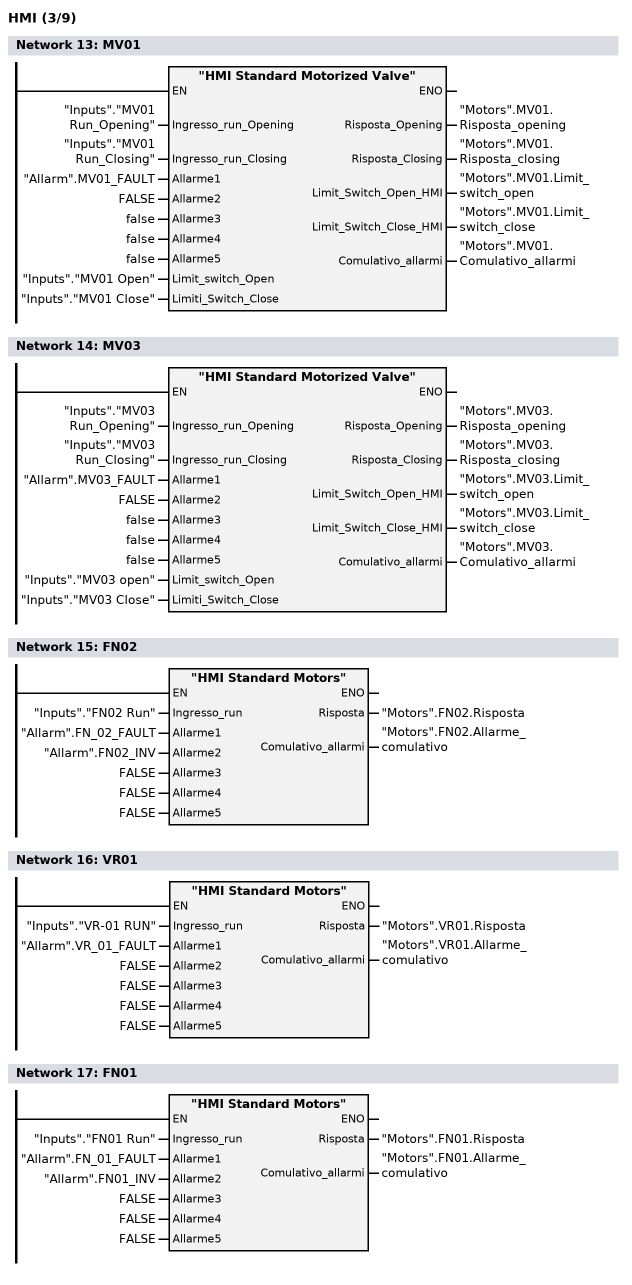
   RUNG wire#powerrail
      "HMI Standard Motorized Valve"(Ingresso_run_Opening := "Inputs"."MV01 Run_Opening", Ingresso_run_Closing := "Inputs"."MV01 Run_Closing", Allarme1 := "Allarm".MV01_FAULT, Allarme2 := FALSE, Allarme3 := false, Allarme4 := false, Allarme5 := false, Limit_switch_Open := "Inputs"."MV01 Open", Limiti_Switch_Close := "Inputs"."MV01 Close", Risposta_Opening => "Motors".MV01.Risposta_opening, Risposta_Closing => "Motors".MV01.Risposta_closing, Limit_Switch_Open_HMI => "Motors".MV01.Limit_switch_open, Limit_Switch_Close_HMI => "Motors".MV01.Limit_switch_close, Comulativo_allarmi => "Motors".MV01.Comulativo_allarmi)
   END_RUNG
   // the same network as SCL:
   "HMI Standard Motorized Valve"(Ingresso_run_Opening := "Inputs"."MV01 Run_Opening",
                           Ingresso_run_Closing := "Inputs"."MV01 Run_Closing",
                           Allarme1 := "Allarm".MV01_FAULT,
                           Allarme2 := FALSE,
                           Allarme3 := false,
                           Allarme4 := false,
                           Allarme5 := false,
                           Limit_switch_Open := "Inputs"."MV01 Open",
                           Limiti_Switch_Close := "Inputs"."MV01 Close",
                           Risposta_Opening => "Motors".MV01.Risposta_opening,
                           Risposta_Closing => "Motors".MV01.Risposta_closing,
                           Limit_Switch_Open_HMI => "Motors".MV01.Limit_switch_open,
                           Limit_Switch_Close_HMI => "Motors".MV01.Limit_switch_close,
                           Comulativo_allarmi => "Motors".MV01.Comulativo_allarmi);
END_REGION

REGION Network 14: MV03
   RUNG wire#powerrail
      "HMI Standard Motorized Valve"(Ingresso_run_Opening := "Inputs"."MV03 Run_Opening", Ingresso_run_Closing := "Inputs"."MV03 Run_Closing", Allarme1 := "Allarm".MV03_FAULT, Allarme2 := FALSE, Allarme3 := false, Allarme4 := false, Allarme5 := false, Limit_switch_Open := "Inputs"."MV03 open", Limiti_Switch_Close := "Inputs"."MV03 Close", Risposta_Opening => "Motors".MV03.Risposta_opening, Risposta_Closing => "Motors".MV03.Risposta_closing, Limit_Switch_Open_HMI => "Motors".MV03.Limit_switch_open, Limit_Switch_Close_HMI => "Motors".MV03.Limit_switch_close, Comulativo_allarmi => "Motors".MV03.Comulativo_allarmi)
   END_RUNG
   // the same network as SCL:
   "HMI Standard Motorized Valve"(Ingresso_run_Opening := "Inputs"."MV03 Run_Opening",
                           Ingresso_run_Closing := "Inputs"."MV03 Run_Closing",
                           Allarme1 := "Allarm".MV03_FAULT,
                           Allarme2 := FALSE,
                           Allarme3 := false,
                           Allarme4 := false,
                           Allarme5 := false,
                           Limit_switch_Open := "Inputs"."MV03 open",
                           Limiti_Switch_Close := "Inputs"."MV03 Close",
                           Risposta_Opening => "Motors".MV03.Risposta_opening,
                           Risposta_Closing => "Motors".MV03.Risposta_closing,
                           Limit_Switch_Open_HMI => "Motors".MV03.Limit_switch_open,
                           Limit_Switch_Close_HMI => "Motors".MV03.Limit_switch_close,
                           Comulativo_allarmi => "Motors".MV03.Comulativo_allarmi);
END_REGION

REGION Network 15: FN02
   RUNG wire#powerrail
      "HMI Standard Motors"(Ingresso_run := "Inputs"."FN02 Run", Allarme1 := "Allarm".FN_02_FAULT, Allarme2 := "Allarm".FN02_INV, Allarme3 := FALSE, Allarme4 := FALSE, Allarme5 := FALSE, Risposta => "Motors".FN02.Risposta, Comulativo_allarmi => "Motors".FN02.Allarme_comulativo)
   END_RUNG
   // the same network as SCL:
   "HMI Standard Motors"(Ingresso_run := "Inputs"."FN02 Run",
                         Allarme1 := "Allarm".FN_02_FAULT,
                         Allarme2 := "Allarm".FN02_INV,
                         Allarme3 := FALSE,
                         Allarme4 := FALSE,
                         Allarme5 := FALSE,
                         Risposta => "Motors".FN02.Risposta,
                         Comulativo_allarmi => "Motors".FN02.Allarme_comulativo);
END_REGION

REGION Network 16: VR01
   RUNG wire#powerrail
      "HMI Standard Motors"(Ingresso_run := "Inputs"."VR-01 RUN", Allarme1 := "Allarm".VR_01_FAULT, Allarme2 := FALSE, Allarme3 := FALSE, Allarme4 := FALSE, Allarme5 := FALSE, Risposta => "Motors".VR01.Risposta, Comulativo_allarmi => "Motors".VR01.Allarme_comulativo)
   END_RUNG
   // the same network as SCL:
   "HMI Standard Motors"(Ingresso_run := "Inputs"."VR-01 RUN",
                         Allarme1 := "Allarm".VR_01_FAULT,
                         Allarme2 := FALSE,
                         Allarme3 := FALSE,
                         Allarme4 := FALSE,
                         Allarme5 := FALSE,
                         Risposta => "Motors".VR01.Risposta,
                         Comulativo_allarmi => "Motors".VR01.Allarme_comulativo);
END_REGION

REGION Network 17: FN01
   RUNG wire#powerrail
      "HMI Standard Motors"(Ingresso_run := "Inputs"."FN01 Run", Allarme1 := "Allarm".FN_01_FAULT, Allarme2 := "Allarm".FN01_INV, Allarme3 := FALSE, Allarme4 := FALSE, Allarme5 := FALSE, Risposta => "Motors".FN01.Risposta, Comulativo_allarmi => "Motors".FN01.Allarme_comulativo)
   END_RUNG
   // the same network as SCL:
   "HMI Standard Motors"(Ingresso_run := "Inputs"."FN01 Run",
                         Allarme1 := "Allarm".FN_01_FAULT,
                         Allarme2 := "Allarm".FN01_INV,
                         Allarme3 := FALSE,
                         Allarme4 := FALSE,
                         Allarme5 := FALSE,
                         Risposta => "Motors".FN01.Risposta,
                         Comulativo_allarmi => "Motors".FN01.Allarme_comulativo);
END_REGION

REGION Network 18: VR02
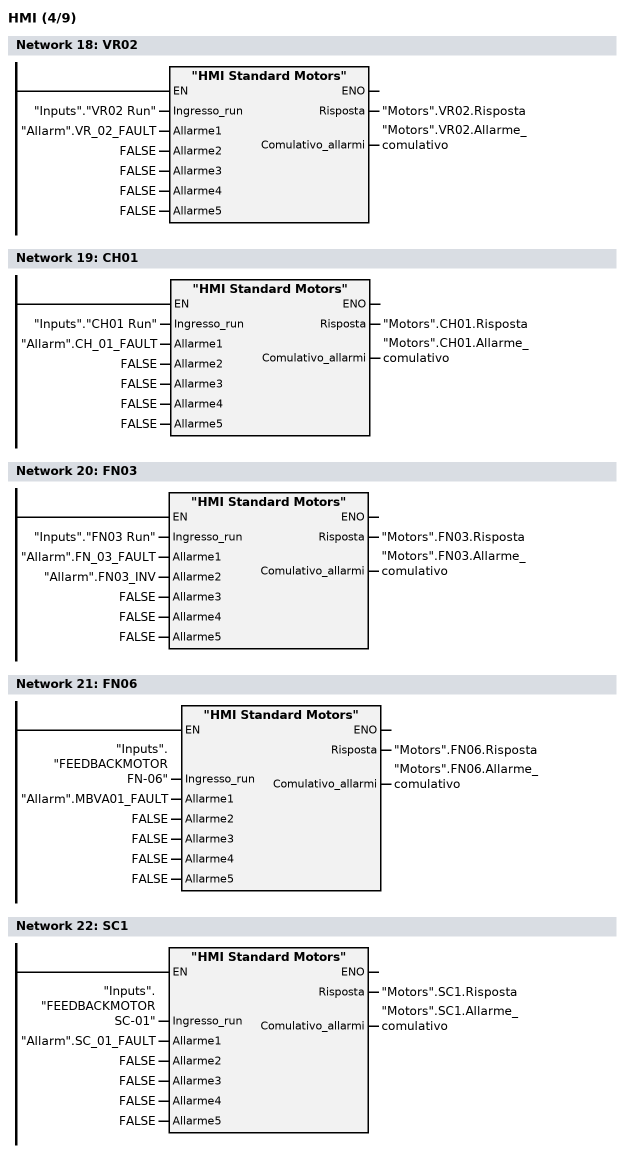
   RUNG wire#powerrail
      "HMI Standard Motors"(Ingresso_run := "Inputs"."VR02 Run", Allarme1 := "Allarm".VR_02_FAULT, Allarme2 := FALSE, Allarme3 := FALSE, Allarme4 := FALSE, Allarme5 := FALSE, Risposta => "Motors".VR02.Risposta, Comulativo_allarmi => "Motors".VR02.Allarme_comulativo)
   END_RUNG
   // the same network as SCL:
   "HMI Standard Motors"(Ingresso_run := "Inputs"."VR02 Run",
                         Allarme1 := "Allarm".VR_02_FAULT,
                         Allarme2 := FALSE,
                         Allarme3 := FALSE,
                         Allarme4 := FALSE,
                         Allarme5 := FALSE,
                         Risposta => "Motors".VR02.Risposta,
                         Comulativo_allarmi => "Motors".VR02.Allarme_comulativo);
END_REGION

REGION Network 19: CH01
   RUNG wire#powerrail
      "HMI Standard Motors"(Ingresso_run := "Inputs"."CH01 Run", Allarme1 := "Allarm".CH_01_FAULT, Allarme2 := FALSE, Allarme3 := FALSE, Allarme4 := FALSE, Allarme5 := FALSE, Risposta => "Motors".CH01.Risposta, Comulativo_allarmi => "Motors".CH01.Allarme_comulativo)
   END_RUNG
   // the same network as SCL:
   "HMI Standard Motors"(Ingresso_run := "Inputs"."CH01 Run",
                         Allarme1 := "Allarm".CH_01_FAULT,
                         Allarme2 := FALSE,
                         Allarme3 := FALSE,
                         Allarme4 := FALSE,
                         Allarme5 := FALSE,
                         Risposta => "Motors".CH01.Risposta,
                         Comulativo_allarmi => "Motors".CH01.Allarme_comulativo);
END_REGION

REGION Network 20: FN03
   RUNG wire#powerrail
      "HMI Standard Motors"(Ingresso_run := "Inputs"."FN03 Run", Allarme1 := "Allarm".FN_03_FAULT, Allarme2 := "Allarm".FN03_INV, Allarme3 := FALSE, Allarme4 := FALSE, Allarme5 := FALSE, Risposta => "Motors".FN03.Risposta, Comulativo_allarmi => "Motors".FN03.Allarme_comulativo)
   END_RUNG
   // the same network as SCL:
   "HMI Standard Motors"(Ingresso_run := "Inputs"."FN03 Run",
                         Allarme1 := "Allarm".FN_03_FAULT,
                         Allarme2 := "Allarm".FN03_INV,
                         Allarme3 := FALSE,
                         Allarme4 := FALSE,
                         Allarme5 := FALSE,
                         Risposta => "Motors".FN03.Risposta,
                         Comulativo_allarmi => "Motors".FN03.Allarme_comulativo);
END_REGION

REGION Network 21: FN06
   RUNG wire#powerrail
      "HMI Standard Motors"(Ingresso_run := "Inputs"."FEEDBACKMOTOR FN-06", Allarme1 := "Allarm".MBVA01_FAULT, Allarme2 := FALSE, Allarme3 := FALSE, Allarme4 := FALSE, Allarme5 := FALSE, Risposta => "Motors".FN06.Risposta, Comulativo_allarmi => "Motors".FN06.Allarme_comulativo)
   END_RUNG
   // the same network as SCL:
   "HMI Standard Motors"(Ingresso_run := "Inputs"."FEEDBACKMOTOR FN-06",
                         Allarme1 := "Allarm".MBVA01_FAULT,
                         Allarme2 := FALSE,
                         Allarme3 := FALSE,
                         Allarme4 := FALSE,
                         Allarme5 := FALSE,
                         Risposta => "Motors".FN06.Risposta,
                         Comulativo_allarmi => "Motors".FN06.Allarme_comulativo);
END_REGION

REGION Network 22: SC1
   RUNG wire#powerrail
      "HMI Standard Motors"(Ingresso_run := "Inputs"."FEEDBACKMOTOR SC-01", Allarme1 := "Allarm".SC_01_FAULT, Allarme2 := FALSE, Allarme3 := FALSE, Allarme4 := FALSE, Allarme5 := FALSE, Risposta => "Motors".SC1.Risposta, Comulativo_allarmi => "Motors".SC1.Allarme_comulativo)
   END_RUNG
   // the same network as SCL:
   "HMI Standard Motors"(Ingresso_run := "Inputs"."FEEDBACKMOTOR SC-01",
                         Allarme1 := "Allarm".SC_01_FAULT,
                         Allarme2 := FALSE,
                         Allarme3 := FALSE,
                         Allarme4 := FALSE,
                         Allarme5 := FALSE,
                         Risposta => "Motors".SC1.Risposta,
                         Comulativo_allarmi => "Motors".SC1.Allarme_comulativo);
END_REGION

REGION Network 23: FN01 FAN DELETED
END_REGION

REGION Network 24: LD01 MF
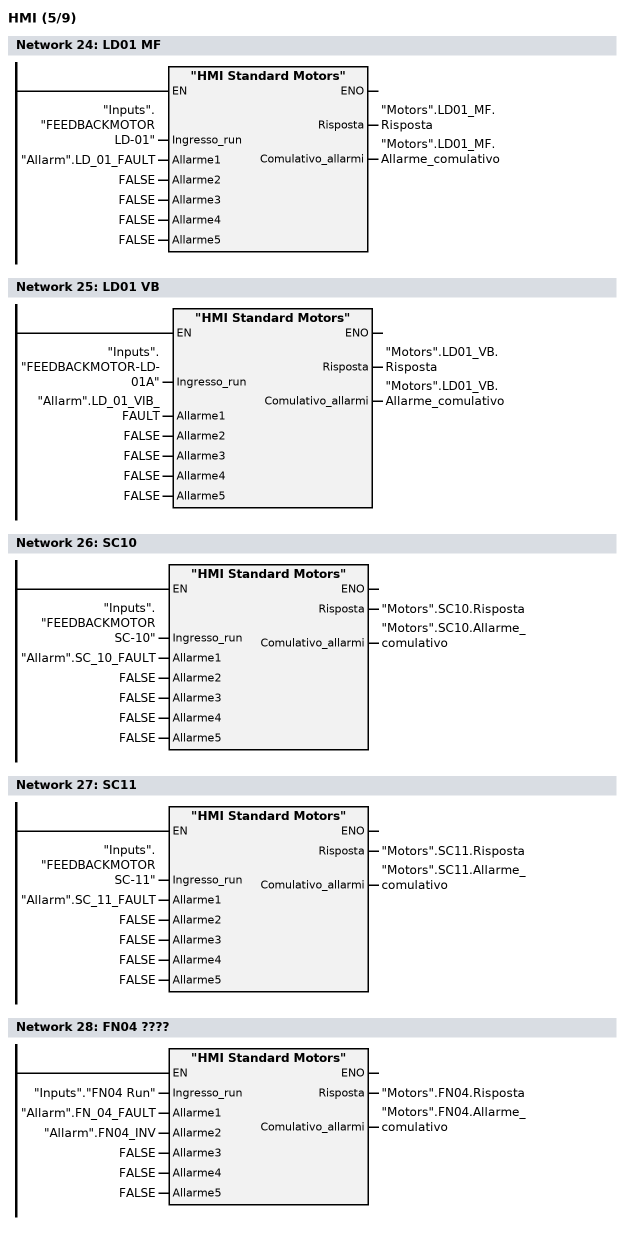
   RUNG wire#powerrail
      "HMI Standard Motors"(Ingresso_run := "Inputs"."FEEDBACKMOTOR LD-01", Allarme1 := "Allarm".LD_01_FAULT, Allarme2 := FALSE, Allarme3 := FALSE, Allarme4 := FALSE, Allarme5 := FALSE, Risposta => "Motors".LD01_MF.Risposta, Comulativo_allarmi => "Motors".LD01_MF.Allarme_comulativo)
   END_RUNG
   // the same network as SCL:
   "HMI Standard Motors"(Ingresso_run := "Inputs"."FEEDBACKMOTOR LD-01",
                         Allarme1 := "Allarm".LD_01_FAULT,
                         Allarme2 := FALSE,
                         Allarme3 := FALSE,
                         Allarme4 := FALSE,
                         Allarme5 := FALSE,
                         Risposta => "Motors".LD01_MF.Risposta,
                         Comulativo_allarmi => "Motors".LD01_MF.Allarme_comulativo);
END_REGION

REGION Network 25: LD01 VB
   RUNG wire#powerrail
      "HMI Standard Motors"(Ingresso_run := "Inputs"."FEEDBACKMOTOR-LD-01A", Allarme1 := "Allarm".LD_01_VIB_FAULT, Allarme2 := FALSE, Allarme3 := FALSE, Allarme4 := FALSE, Allarme5 := FALSE, Risposta => "Motors".LD01_VB.Risposta, Comulativo_allarmi => "Motors".LD01_VB.Allarme_comulativo)
   END_RUNG
   // the same network as SCL:
   "HMI Standard Motors"(Ingresso_run := "Inputs"."FEEDBACKMOTOR-LD-01A",
                         Allarme1 := "Allarm".LD_01_VIB_FAULT,
                         Allarme2 := FALSE,
                         Allarme3 := FALSE,
                         Allarme4 := FALSE,
                         Allarme5 := FALSE,
                         Risposta => "Motors".LD01_VB.Risposta,
                         Comulativo_allarmi => "Motors".LD01_VB.Allarme_comulativo);
END_REGION

REGION Network 26: SC10
   RUNG wire#powerrail
      "HMI Standard Motors"(Ingresso_run := "Inputs"."FEEDBACKMOTOR SC-10", Allarme1 := "Allarm".SC_10_FAULT, Allarme2 := FALSE, Allarme3 := FALSE, Allarme4 := FALSE, Allarme5 := FALSE, Risposta => "Motors".SC10.Risposta, Comulativo_allarmi => "Motors".SC10.Allarme_comulativo)
   END_RUNG
   // the same network as SCL:
   "HMI Standard Motors"(Ingresso_run := "Inputs"."FEEDBACKMOTOR SC-10",
                         Allarme1 := "Allarm".SC_10_FAULT,
                         Allarme2 := FALSE,
                         Allarme3 := FALSE,
                         Allarme4 := FALSE,
                         Allarme5 := FALSE,
                         Risposta => "Motors".SC10.Risposta,
                         Comulativo_allarmi => "Motors".SC10.Allarme_comulativo);
END_REGION

REGION Network 27: SC11
   RUNG wire#powerrail
      "HMI Standard Motors"(Ingresso_run := "Inputs"."FEEDBACKMOTOR SC-11", Allarme1 := "Allarm".SC_11_FAULT, Allarme2 := FALSE, Allarme3 := FALSE, Allarme4 := FALSE, Allarme5 := FALSE, Risposta => "Motors".SC11.Risposta, Comulativo_allarmi => "Motors".SC11.Allarme_comulativo)
   END_RUNG
   // the same network as SCL:
   "HMI Standard Motors"(Ingresso_run := "Inputs"."FEEDBACKMOTOR SC-11",
                         Allarme1 := "Allarm".SC_11_FAULT,
                         Allarme2 := FALSE,
                         Allarme3 := FALSE,
                         Allarme4 := FALSE,
                         Allarme5 := FALSE,
                         Risposta => "Motors".SC11.Risposta,
                         Comulativo_allarmi => "Motors".SC11.Allarme_comulativo);
END_REGION

REGION Network 28: FN04 ????
   RUNG wire#powerrail
      "HMI Standard Motors"(Ingresso_run := "Inputs"."FN04 Run", Allarme1 := "Allarm".FN_04_FAULT, Allarme2 := "Allarm".FN04_INV, Allarme3 := FALSE, Allarme4 := FALSE, Allarme5 := FALSE, Risposta => "Motors".FN04.Risposta, Comulativo_allarmi => "Motors".FN04.Allarme_comulativo)
   END_RUNG
   // the same network as SCL:
   "HMI Standard Motors"(Ingresso_run := "Inputs"."FN04 Run",
                         Allarme1 := "Allarm".FN_04_FAULT,
                         Allarme2 := "Allarm".FN04_INV,
                         Allarme3 := FALSE,
                         Allarme4 := FALSE,
                         Allarme5 := FALSE,
                         Risposta => "Motors".FN04.Risposta,
                         Comulativo_allarmi => "Motors".FN04.Allarme_comulativo);
END_REGION

REGION Network 29: VR03
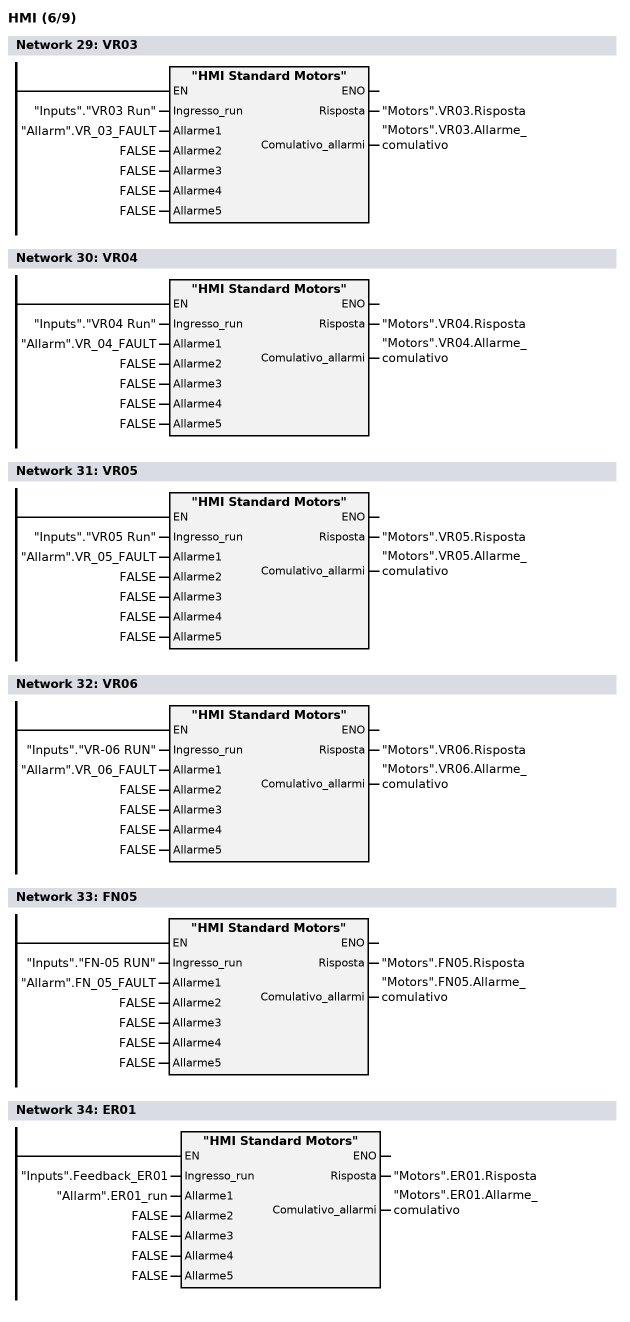
   RUNG wire#powerrail
      "HMI Standard Motors"(Ingresso_run := "Inputs"."VR03 Run", Allarme1 := "Allarm".VR_03_FAULT, Allarme2 := FALSE, Allarme3 := FALSE, Allarme4 := FALSE, Allarme5 := FALSE, Risposta => "Motors".VR03.Risposta, Comulativo_allarmi => "Motors".VR03.Allarme_comulativo)
   END_RUNG
   // the same network as SCL:
   "HMI Standard Motors"(Ingresso_run := "Inputs"."VR03 Run",
                         Allarme1 := "Allarm".VR_03_FAULT,
                         Allarme2 := FALSE,
                         Allarme3 := FALSE,
                         Allarme4 := FALSE,
                         Allarme5 := FALSE,
                         Risposta => "Motors".VR03.Risposta,
                         Comulativo_allarmi => "Motors".VR03.Allarme_comulativo);
END_REGION

REGION Network 30: VR04
   RUNG wire#powerrail
      "HMI Standard Motors"(Ingresso_run := "Inputs"."VR04 Run", Allarme1 := "Allarm".VR_04_FAULT, Allarme2 := FALSE, Allarme3 := FALSE, Allarme4 := FALSE, Allarme5 := FALSE, Risposta => "Motors".VR04.Risposta, Comulativo_allarmi => "Motors".VR04.Allarme_comulativo)
   END_RUNG
   // the same network as SCL:
   "HMI Standard Motors"(Ingresso_run := "Inputs"."VR04 Run",
                         Allarme1 := "Allarm".VR_04_FAULT,
                         Allarme2 := FALSE,
                         Allarme3 := FALSE,
                         Allarme4 := FALSE,
                         Allarme5 := FALSE,
                         Risposta => "Motors".VR04.Risposta,
                         Comulativo_allarmi => "Motors".VR04.Allarme_comulativo);
END_REGION

REGION Network 31: VR05
   RUNG wire#powerrail
      "HMI Standard Motors"(Ingresso_run := "Inputs"."VR05 Run", Allarme1 := "Allarm".VR_05_FAULT, Allarme2 := FALSE, Allarme3 := FALSE, Allarme4 := FALSE, Allarme5 := FALSE, Risposta => "Motors".VR05.Risposta, Comulativo_allarmi => "Motors".VR05.Allarme_comulativo)
   END_RUNG
   // the same network as SCL:
   "HMI Standard Motors"(Ingresso_run := "Inputs"."VR05 Run",
                         Allarme1 := "Allarm".VR_05_FAULT,
                         Allarme2 := FALSE,
                         Allarme3 := FALSE,
                         Allarme4 := FALSE,
                         Allarme5 := FALSE,
                         Risposta => "Motors".VR05.Risposta,
                         Comulativo_allarmi => "Motors".VR05.Allarme_comulativo);
END_REGION

REGION Network 32: VR06
   RUNG wire#powerrail
      "HMI Standard Motors"(Ingresso_run := "Inputs"."VR-06 RUN", Allarme1 := "Allarm".VR_06_FAULT, Allarme2 := FALSE, Allarme3 := FALSE, Allarme4 := FALSE, Allarme5 := FALSE, Risposta => "Motors".VR06.Risposta, Comulativo_allarmi => "Motors".VR06.Allarme_comulativo)
   END_RUNG
   // the same network as SCL:
   "HMI Standard Motors"(Ingresso_run := "Inputs"."VR-06 RUN",
                         Allarme1 := "Allarm".VR_06_FAULT,
                         Allarme2 := FALSE,
                         Allarme3 := FALSE,
                         Allarme4 := FALSE,
                         Allarme5 := FALSE,
                         Risposta => "Motors".VR06.Risposta,
                         Comulativo_allarmi => "Motors".VR06.Allarme_comulativo);
END_REGION

REGION Network 33: FN05
   RUNG wire#powerrail
      "HMI Standard Motors"(Ingresso_run := "Inputs"."FN-05 RUN", Allarme1 := "Allarm".FN_05_FAULT, Allarme2 := FALSE, Allarme3 := FALSE, Allarme4 := FALSE, Allarme5 := FALSE, Risposta => "Motors".FN05.Risposta, Comulativo_allarmi => "Motors".FN05.Allarme_comulativo)
   END_RUNG
   // the same network as SCL:
   "HMI Standard Motors"(Ingresso_run := "Inputs"."FN-05 RUN",
                         Allarme1 := "Allarm".FN_05_FAULT,
                         Allarme2 := FALSE,
                         Allarme3 := FALSE,
                         Allarme4 := FALSE,
                         Allarme5 := FALSE,
                         Risposta => "Motors".FN05.Risposta,
                         Comulativo_allarmi => "Motors".FN05.Allarme_comulativo);
END_REGION

REGION Network 34: ER01
   RUNG wire#powerrail
      "HMI Standard Motors"(Ingresso_run := "Inputs".Feedback_ER01, Allarme1 := "Allarm".ER01_run, Allarme2 := FALSE, Allarme3 := FALSE, Allarme4 := FALSE, Allarme5 := FALSE, Risposta => "Motors".ER01.Risposta, Comulativo_allarmi => "Motors".ER01.Allarme_comulativo)
   END_RUNG
   // the same network as SCL:
   "HMI Standard Motors"(Ingresso_run := "Inputs".Feedback_ER01,
                         Allarme1 := "Allarm".ER01_run,
                         Allarme2 := FALSE,
                         Allarme3 := FALSE,
                         Allarme4 := FALSE,
                         Allarme5 := FALSE,
                         Risposta => "Motors".ER01.Risposta,
                         Comulativo_allarmi => "Motors".ER01.Allarme_comulativo);
END_REGION

REGION Network 35: PV14
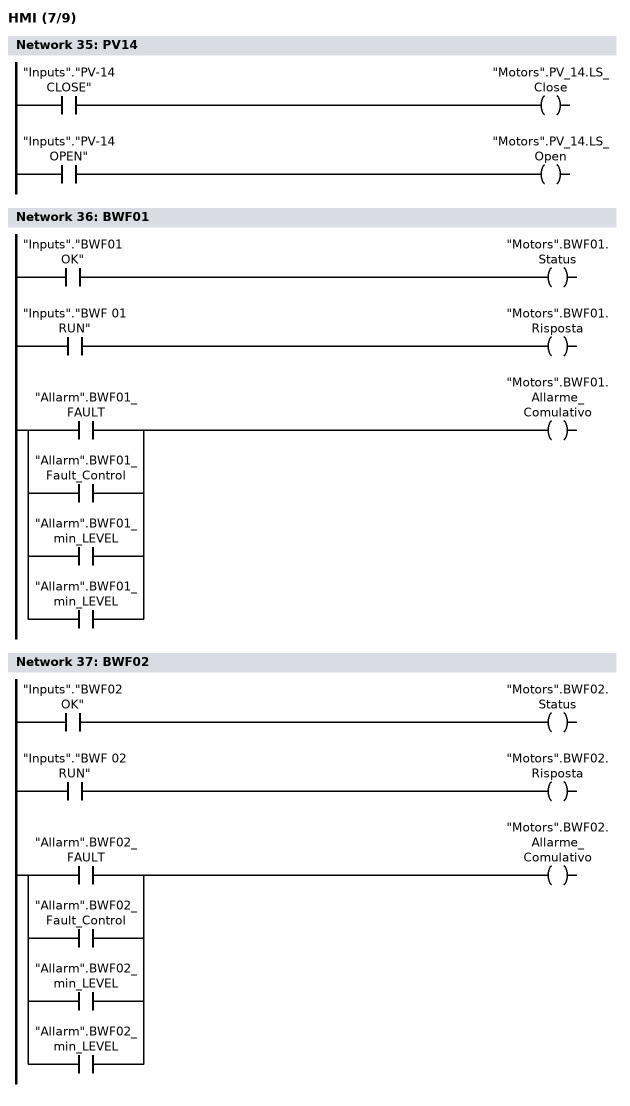
   RUNG wire#powerrail
      Contact( "Inputs"."PV-14 CLOSE" )
      Coil( "Motors".PV_14.LS_Close )
   END_RUNG
   RUNG wire#powerrail
      Contact( "Inputs"."PV-14 OPEN" )
      Coil( "Motors".PV_14.LS_Open )
   END_RUNG
   // the same network as SCL:
   "Motors".PV_14.LS_Close := "Inputs"."PV-14 CLOSE";
   "Motors".PV_14.LS_Open := "Inputs"."PV-14 OPEN";
END_REGION

REGION Network 36: BWF01
   RUNG wire#powerrail
      Contact( "Inputs"."BWF01 OK" )
      Coil( "Motors".BWF01.Status )
   END_RUNG
   RUNG wire#powerrail
      Contact( "Inputs"."BWF 01 RUN" )
      Coil( "Motors".BWF01.Risposta )
   END_RUNG
   RUNG wire#powerrail
      Contact( "Allarm".BWF01_FAULT )
      wire#w1
      Coil( "Motors".BWF01.Allarme_Comulativo )
   END_RUNG
   RUNG wire#powerrail
      Contact( "Allarm".BWF01_Fault_Control )
   END_RUNG wire#w1
   RUNG wire#powerrail
      Contact( "Allarm".BWF01_min_LEVEL )
   END_RUNG wire#w1
   RUNG wire#powerrail
      Contact( "Allarm".BWF01_min_LEVEL )
   END_RUNG wire#w1
   // the same network as SCL:
   "Motors".BWF01.Status := "Inputs"."BWF01 OK";
   "Motors".BWF01.Risposta := "Inputs"."BWF 01 RUN";
   "Motors".BWF01.Allarme_Comulativo := "Allarm".BWF01_FAULT OR "Allarm".BWF01_Fault_Control OR "Allarm".BWF01_min_LEVEL OR "Allarm".BWF01_min_LEVEL;
END_REGION

REGION Network 37: BWF02
   RUNG wire#powerrail
      Contact( "Inputs"."BWF02 OK" )
      Coil( "Motors".BWF02.Status )
   END_RUNG
   RUNG wire#powerrail
      Contact( "Inputs"."BWF 02 RUN" )
      Coil( "Motors".BWF02.Risposta )
   END_RUNG
   RUNG wire#powerrail
      Contact( "Allarm".BWF02_FAULT )
      wire#w1
      Coil( "Motors".BWF02.Allarme_Comulativo )
   END_RUNG
   RUNG wire#powerrail
      Contact( "Allarm".BWF02_Fault_Control )
   END_RUNG wire#w1
   RUNG wire#powerrail
      Contact( "Allarm".BWF02_min_LEVEL )
   END_RUNG wire#w1
   RUNG wire#powerrail
      Contact( "Allarm".BWF02_min_LEVEL )
   END_RUNG wire#w1
   // the same network as SCL:
   "Motors".BWF02.Status := "Inputs"."BWF02 OK";
   "Motors".BWF02.Risposta := "Inputs"."BWF 02 RUN";
   "Motors".BWF02.Allarme_Comulativo := "Allarm".BWF02_FAULT OR "Allarm".BWF02_Fault_Control OR "Allarm".BWF02_min_LEVEL OR "Allarm".BWF02_min_LEVEL;
END_REGION

REGION Network 38: PV01
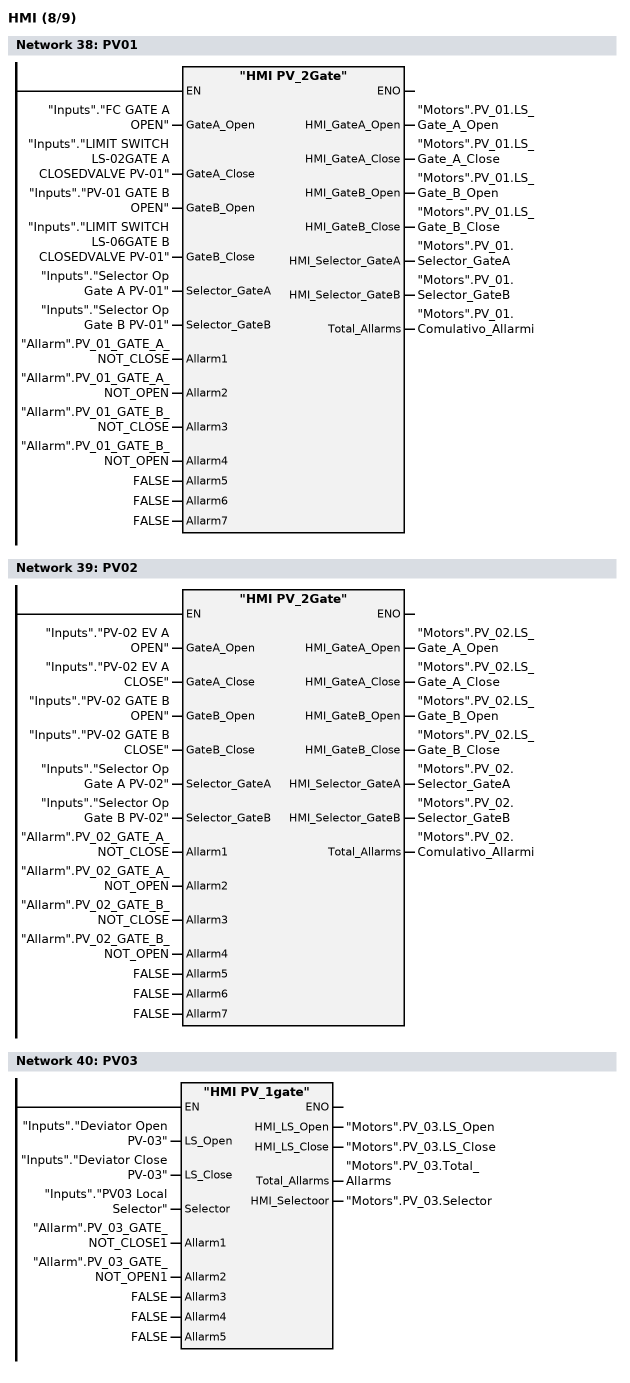
   RUNG wire#powerrail
      "HMI PV_2Gate"(GateA_Open := "Inputs"."FC GATE A OPEN", GateA_Close := "Inputs"."LIMIT SWITCH LS-02GATE A CLOSEDVALVE PV-01", GateB_Open := "Inputs"."PV-01 GATE B OPEN", GateB_Close := "Inputs"."LIMIT SWITCH LS-06GATE B CLOSEDVALVE PV-01", Selector_GateA := "Inputs"."Selector Op Gate A PV-01", Selector_GateB := "Inputs"."Selector Op Gate B PV-01", Allarm1 := "Allarm".PV_01_GATE_A_NOT_CLOSE, Allarm2 := "Allarm".PV_01_GATE_A_NOT_OPEN, Allarm3 := "Allarm".PV_01_GATE_B_NOT_CLOSE, Allarm4 := "Allarm".PV_01_GATE_B_NOT_OPEN, Allarm5 := FALSE, Allarm6 := FALSE, Allarm7 := FALSE, HMI_GateA_Open => "Motors".PV_01.LS_Gate_A_Open, HMI_GateA_Close => "Motors".PV_01.LS_Gate_A_Close, HMI_GateB_Open => "Motors".PV_01.LS_Gate_B_Open, HMI_GateB_Close => "Motors".PV_01.LS_Gate_B_Close, HMI_Selector_GateA => "Motors".PV_01.Selector_GateA, HMI_Selector_GateB => "Motors".PV_01.Selector_GateB, Total_Allarms => "Motors".PV_01.Comulativo_Allarmi)
   END_RUNG
   // the same network as SCL:
   "HMI PV_2Gate"(GateA_Open := "Inputs"."FC GATE A OPEN",
                  GateA_Close := "Inputs"."LIMIT SWITCH LS-02GATE A CLOSEDVALVE PV-01",
                  GateB_Open := "Inputs"."PV-01 GATE B OPEN",
                  GateB_Close := "Inputs"."LIMIT SWITCH LS-06GATE B CLOSEDVALVE PV-01",
                  Selector_GateA := "Inputs"."Selector Op Gate A PV-01",
                  Selector_GateB := "Inputs"."Selector Op Gate B PV-01",
                  Allarm1 := "Allarm".PV_01_GATE_A_NOT_CLOSE,
                  Allarm2 := "Allarm".PV_01_GATE_A_NOT_OPEN,
                  Allarm3 := "Allarm".PV_01_GATE_B_NOT_CLOSE,
                  Allarm4 := "Allarm".PV_01_GATE_B_NOT_OPEN,
                  Allarm5 := FALSE,
                  Allarm6 := FALSE,
                  Allarm7 := FALSE,
                  HMI_GateA_Open => "Motors".PV_01.LS_Gate_A_Open,
                  HMI_GateA_Close => "Motors".PV_01.LS_Gate_A_Close,
                  HMI_GateB_Open => "Motors".PV_01.LS_Gate_B_Open,
                  HMI_GateB_Close => "Motors".PV_01.LS_Gate_B_Close,
                  HMI_Selector_GateA => "Motors".PV_01.Selector_GateA,
                  HMI_Selector_GateB => "Motors".PV_01.Selector_GateB,
                  Total_Allarms => "Motors".PV_01.Comulativo_Allarmi);
END_REGION

REGION Network 39: PV02
   RUNG wire#powerrail
      "HMI PV_2Gate"(GateA_Open := "Inputs"."PV-02 EV A OPEN", GateA_Close := "Inputs"."PV-02 EV A CLOSE", GateB_Open := "Inputs"."PV-02 GATE B OPEN", GateB_Close := "Inputs"."PV-02 GATE B CLOSE", Selector_GateA := "Inputs"."Selector Op Gate A PV-02", Selector_GateB := "Inputs"."Selector Op Gate B PV-02", Allarm1 := "Allarm".PV_02_GATE_A_NOT_CLOSE, Allarm2 := "Allarm".PV_02_GATE_A_NOT_OPEN, Allarm3 := "Allarm".PV_02_GATE_B_NOT_CLOSE, Allarm4 := "Allarm".PV_02_GATE_B_NOT_OPEN, Allarm5 := FALSE, Allarm6 := FALSE, Allarm7 := FALSE, HMI_GateA_Open => "Motors".PV_02.LS_Gate_A_Open, HMI_GateA_Close => "Motors".PV_02.LS_Gate_A_Close, HMI_GateB_Open => "Motors".PV_02.LS_Gate_B_Open, HMI_GateB_Close => "Motors".PV_02.LS_Gate_B_Close, HMI_Selector_GateA => "Motors".PV_02.Selector_GateA, HMI_Selector_GateB => "Motors".PV_02.Selector_GateB, Total_Allarms => "Motors".PV_02.Comulativo_Allarmi)
   END_RUNG
   // the same network as SCL:
   "HMI PV_2Gate"(GateA_Open := "Inputs"."PV-02 EV A OPEN",
                  GateA_Close := "Inputs"."PV-02 EV A CLOSE",
                  GateB_Open := "Inputs"."PV-02 GATE B OPEN",
                  GateB_Close := "Inputs"."PV-02 GATE B CLOSE",
                  Selector_GateA := "Inputs"."Selector Op Gate A PV-02",
                  Selector_GateB := "Inputs"."Selector Op Gate B PV-02",
                  Allarm1 := "Allarm".PV_02_GATE_A_NOT_CLOSE,
                  Allarm2 := "Allarm".PV_02_GATE_A_NOT_OPEN,
                  Allarm3 := "Allarm".PV_02_GATE_B_NOT_CLOSE,
                  Allarm4 := "Allarm".PV_02_GATE_B_NOT_OPEN,
                  Allarm5 := FALSE,
                  Allarm6 := FALSE,
                  Allarm7 := FALSE,
                  HMI_GateA_Open => "Motors".PV_02.LS_Gate_A_Open,
                  HMI_GateA_Close => "Motors".PV_02.LS_Gate_A_Close,
                  HMI_GateB_Open => "Motors".PV_02.LS_Gate_B_Open,
                  HMI_GateB_Close => "Motors".PV_02.LS_Gate_B_Close,
                  HMI_Selector_GateA => "Motors".PV_02.Selector_GateA,
                  HMI_Selector_GateB => "Motors".PV_02.Selector_GateB,
                  Total_Allarms => "Motors".PV_02.Comulativo_Allarmi);
END_REGION

REGION Network 40: PV03
   RUNG wire#powerrail
      "HMI PV_1gate"(LS_Open := "Inputs"."Deviator Open PV-03", LS_Close := "Inputs"."Deviator Close PV-03", Selector := "Inputs"."PV03 Local Selector", Allarm1 := "Allarm".PV_03_GATE_NOT_CLOSE1, Allarm2 := "Allarm".PV_03_GATE_NOT_OPEN1, Allarm3 := FALSE, Allarm4 := FALSE, Allarm5 := FALSE, HMI_LS_Open => "Motors".PV_03.LS_Open, HMI_LS_Close => "Motors".PV_03.LS_Close, Total_Allarms => "Motors".PV_03.Total_Allarms, HMI_Selectoor => "Motors".PV_03.Selector)
   END_RUNG
   // the same network as SCL:
   "HMI PV_1gate"(LS_Open := "Inputs"."Deviator Open PV-03",
                  LS_Close := "Inputs"."Deviator Close PV-03",
                  Selector := "Inputs"."PV03 Local Selector",
                  Allarm1 := "Allarm".PV_03_GATE_NOT_CLOSE1,
                  Allarm2 := "Allarm".PV_03_GATE_NOT_OPEN1,
                  Allarm3 := FALSE,
                  Allarm4 := FALSE,
                  Allarm5 := FALSE,
                  HMI_LS_Open => "Motors".PV_03.LS_Open,
                  HMI_LS_Close => "Motors".PV_03.LS_Close,
                  Total_Allarms => "Motors".PV_03.Total_Allarms,
                  HMI_Selectoor => "Motors".PV_03.Selector);
END_REGION

REGION Network 41: PV04
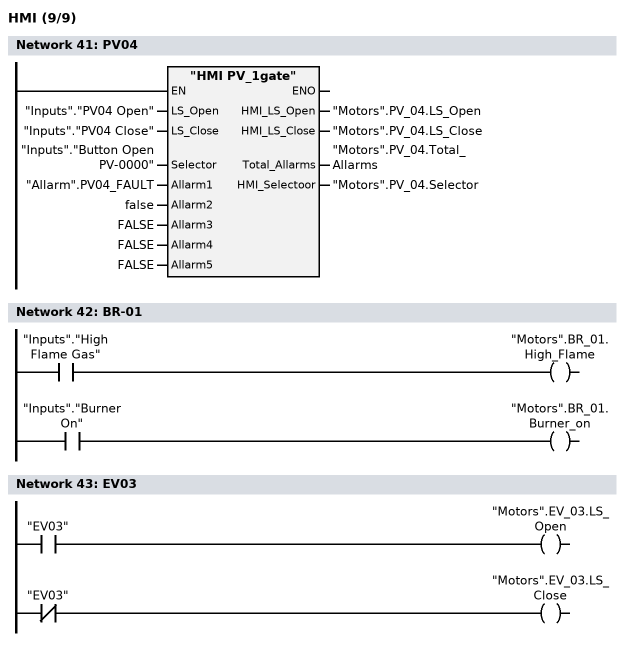
   RUNG wire#powerrail
      "HMI PV_1gate"(LS_Open := "Inputs"."PV04 Open", LS_Close := "Inputs"."PV04 Close", Selector := "Inputs"."Button Open PV-0000", Allarm1 := "Allarm".PV04_FAULT, Allarm2 := false, Allarm3 := FALSE, Allarm4 := FALSE, Allarm5 := FALSE, HMI_LS_Open => "Motors".PV_04.LS_Open, HMI_LS_Close => "Motors".PV_04.LS_Close, Total_Allarms => "Motors".PV_04.Total_Allarms, HMI_Selectoor => "Motors".PV_04.Selector)
   END_RUNG
   // the same network as SCL:
   "HMI PV_1gate"(LS_Open := "Inputs"."PV04 Open",
                  LS_Close := "Inputs"."PV04 Close",
                  Selector := "Inputs"."Button Open PV-0000",
                  Allarm1 := "Allarm".PV04_FAULT,
                  Allarm2 := false,
                  Allarm3 := FALSE,
                  Allarm4 := FALSE,
                  Allarm5 := FALSE,
                  HMI_LS_Open => "Motors".PV_04.LS_Open,
                  HMI_LS_Close => "Motors".PV_04.LS_Close,
                  Total_Allarms => "Motors".PV_04.Total_Allarms,
                  HMI_Selectoor => "Motors".PV_04.Selector);
END_REGION

REGION Network 42: BR-01
   RUNG wire#powerrail
      Contact( "Inputs"."High Flame Gas" )
      Coil( "Motors".BR_01.High_Flame )
   END_RUNG
   RUNG wire#powerrail
      Contact( "Inputs"."Burner On" )
      Coil( "Motors".BR_01.Burner_on )
   END_RUNG
   // the same network as SCL:
   "Motors".BR_01.High_Flame := "Inputs"."High Flame Gas";
   "Motors".BR_01.Burner_on := "Inputs"."Burner On";
END_REGION

REGION Network 43: EV03
   RUNG wire#powerrail
      Contact( "EV03" )
      Coil( "Motors".EV_03.LS_Open )
   END_RUNG
   RUNG wire#powerrail
      I_Contact( "EV03" )
      Coil( "Motors".EV_03.LS_Close )
   END_RUNG
   // the same network as SCL:
   "Motors".EV_03.LS_Open := "EV03";
   "Motors".EV_03.LS_Close := NOT "EV03";
END_REGION
END_FUNCTION

FUNCTION "HMI Inputs" : Void   // FC15, LAD
{ S7_Optimized_Access := 'TRUE' }
VERSION : 0.1
BEGIN

REGION Network 1
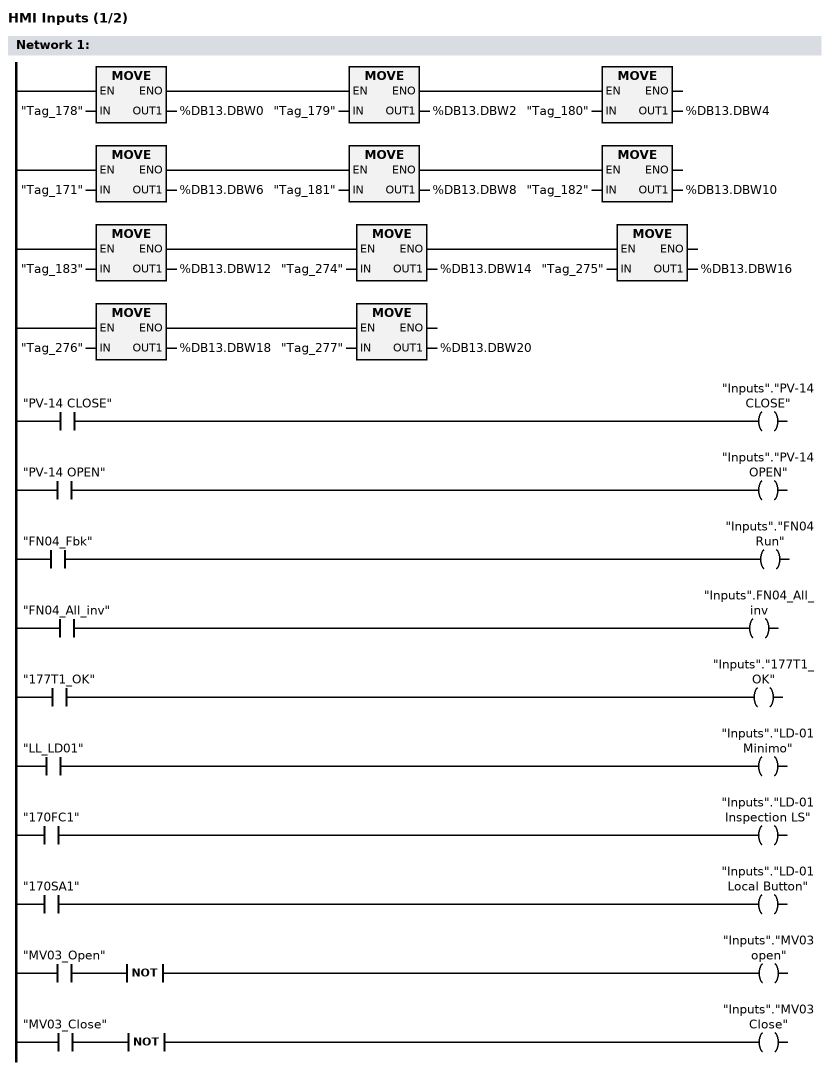
   RUNG wire#powerrail
      Move(in := "Tag_178", out1 => %DB13.DBW0)
      Move(in := "Tag_179", out1 => %DB13.DBW2)
      Move(in := "Tag_180", out1 => %DB13.DBW4)
   END_RUNG
   RUNG wire#powerrail
      Move(in := "Tag_171", out1 => %DB13.DBW6)
      Move(in := "Tag_181", out1 => %DB13.DBW8)
      Move(in := "Tag_182", out1 => %DB13.DBW10)
   END_RUNG
   RUNG wire#powerrail
      Move(in := "Tag_183", out1 => %DB13.DBW12)
      Move(in := "Tag_274", out1 => %DB13.DBW14)
      Move(in := "Tag_275", out1 => %DB13.DBW16)
   END_RUNG
   RUNG wire#powerrail
      Move(in := "Tag_276", out1 => %DB13.DBW18)
      Move(in := "Tag_277", out1 => %DB13.DBW20)
   END_RUNG
   RUNG wire#powerrail
      Contact( "PV-14 CLOSE" )
      Coil( "Inputs"."PV-14 CLOSE" )
   END_RUNG
   RUNG wire#powerrail
      Contact( "PV-14 OPEN" )
      Coil( "Inputs"."PV-14 OPEN" )
   END_RUNG
   RUNG wire#powerrail
      Contact( "FN04_Fbk" )
      Coil( "Inputs"."FN04 Run" )
   END_RUNG
   RUNG wire#powerrail
      Contact( "FN04_All_inv" )
      Coil( "Inputs".FN04_All_inv )
   END_RUNG
   RUNG wire#powerrail
      Contact( "177T1_OK" )
      Coil( "Inputs"."177T1_OK" )
   END_RUNG
   RUNG wire#powerrail
      Contact( "LL_LD01" )
      Coil( "Inputs"."LD-01 Minimo" )
   END_RUNG
   RUNG wire#powerrail
      Contact( "170FC1" )
      Coil( "Inputs"."LD-01 Inspection LS" )
   END_RUNG
   RUNG wire#powerrail
      Contact( "170SA1" )
      Coil( "Inputs"."LD-01 Local Button" )
   END_RUNG
   RUNG wire#powerrail
      Contact( "MV03_Open" )
      Not()
      Coil( "Inputs"."MV03 open" )
   END_RUNG
   RUNG wire#powerrail
      Contact( "MV03_Close" )
      Not()
      Coil( "Inputs"."MV03 Close" )
   END_RUNG
   // the same network as SCL:
   %DB13.DBW0 := "Tag_178";
   %DB13.DBW2 := "Tag_179";
   %DB13.DBW4 := "Tag_180";
   %DB13.DBW6 := "Tag_171";
   %DB13.DBW8 := "Tag_181";
   %DB13.DBW10 := "Tag_182";
   %DB13.DBW12 := "Tag_183";
   %DB13.DBW14 := "Tag_274";
   %DB13.DBW16 := "Tag_275";
   %DB13.DBW18 := "Tag_276";
   %DB13.DBW20 := "Tag_277";
   "Inputs"."PV-14 CLOSE" := "PV-14 CLOSE";
   "Inputs"."PV-14 OPEN" := "PV-14 OPEN";
   "Inputs"."FN04 Run" := "FN04_Fbk";
   "Inputs".FN04_All_inv := "FN04_All_inv";
   "Inputs"."177T1_OK" := "177T1_OK";
   "Inputs"."LD-01 Minimo" := "LL_LD01";
   "Inputs"."LD-01 Inspection LS" := "170FC1";
   "Inputs"."LD-01 Local Button" := "170SA1";
   "Inputs"."MV03 open" := NOT "MV03_Open";
   "Inputs"."MV03 Close" := NOT "MV03_Close";
END_REGION

REGION Network 2: ANALOG
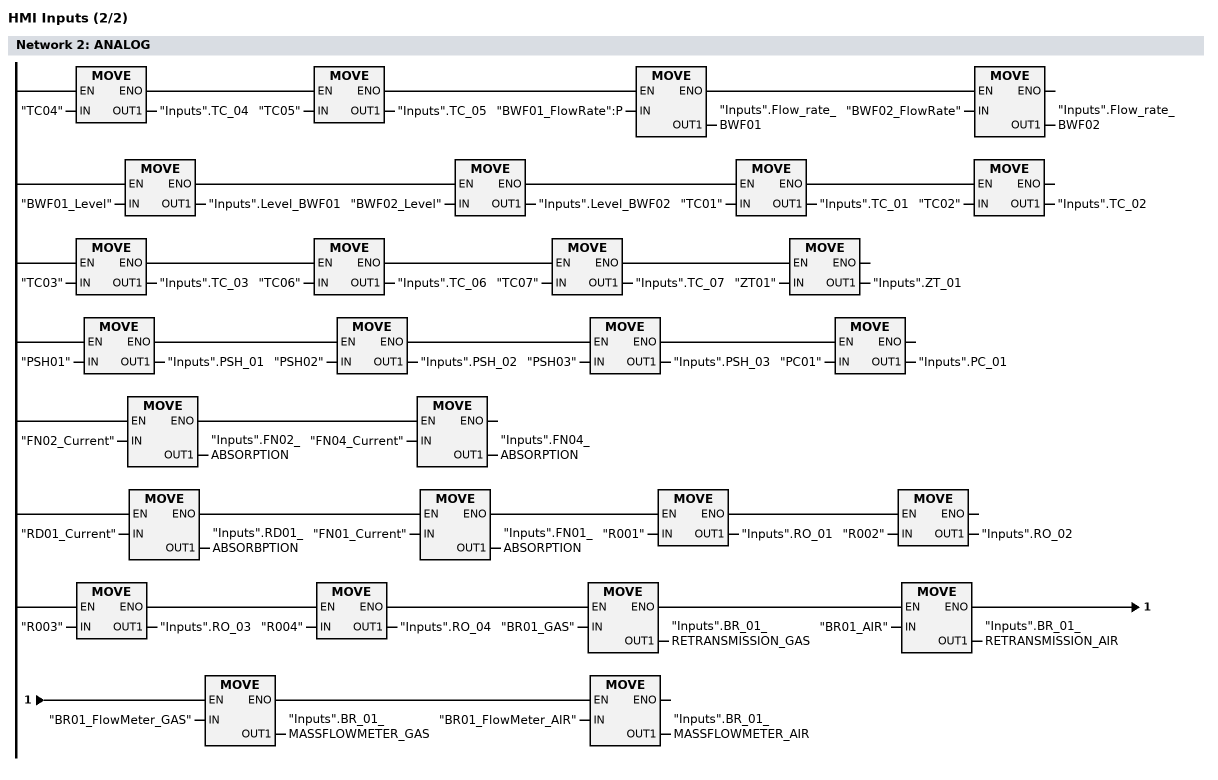
   RUNG wire#powerrail
      Move(in := "TC04", out1 => "Inputs".TC_04)
      Move(in := "TC05", out1 => "Inputs".TC_05)
      Move(in := "BWF01_FlowRate":P, out1 => "Inputs".Flow_rate_BWF01)
      Move(in := "BWF02_FlowRate", out1 => "Inputs".Flow_rate_BWF02)
   END_RUNG
   RUNG wire#powerrail
      Move(in := "BWF01_Level", out1 => "Inputs".Level_BWF01)
      Move(in := "BWF02_Level", out1 => "Inputs".Level_BWF02)
      Move(in := "TC01", out1 => "Inputs".TC_01)
      Move(in := "TC02", out1 => "Inputs".TC_02)
   END_RUNG
   RUNG wire#powerrail
      Move(in := "TC03", out1 => "Inputs".TC_03)
      Move(in := "TC06", out1 => "Inputs".TC_06)
      Move(in := "TC07", out1 => "Inputs".TC_07)
      Move(in := "ZT01", out1 => "Inputs".ZT_01)
   END_RUNG
   RUNG wire#powerrail
      Move(in := "PSH01", out1 => "Inputs".PSH_01)
      Move(in := "PSH02", out1 => "Inputs".PSH_02)
      Move(in := "PSH03", out1 => "Inputs".PSH_03)
      Move(in := "PC01", out1 => "Inputs".PC_01)
   END_RUNG
   RUNG wire#powerrail
      Move(in := "FN02_Current", out1 => "Inputs".FN02_ABSORPTION)
      Move(in := "FN04_Current", out1 => "Inputs".FN04_ABSORPTION)
   END_RUNG
   RUNG wire#powerrail
      Move(in := "RD01_Current", out1 => "Inputs".RD01_ABSORBPTION)
      Move(in := "FN01_Current", out1 => "Inputs".FN01_ABSORPTION)
      Move(in := "R001", out1 => "Inputs".RO_01)
      Move(in := "R002", out1 => "Inputs".RO_02)
   END_RUNG
   RUNG wire#powerrail
      Move(in := "R003", out1 => "Inputs".RO_03)
      Move(in := "R004", out1 => "Inputs".RO_04)
      Move(in := "BR01_GAS", out1 => "Inputs".BR_01_RETRANSMISSION_GAS)
      Move(in := "BR01_AIR", out1 => "Inputs".BR_01_RETRANSMISSION_AIR)
      Move(in := "BR01_FlowMeter_GAS", out1 => "Inputs".BR_01_MASSFLOWMETER_GAS)
      Move(in := "BR01_FlowMeter_AIR", out1 => "Inputs".BR_01_MASSFLOWMETER_AIR)
   END_RUNG
   // the same network as SCL:
   "Inputs".TC_04 := "TC04";
   "Inputs".TC_05 := "TC05";
   "Inputs".Flow_rate_BWF01 := "BWF01_FlowRate":P;
   "Inputs".Flow_rate_BWF02 := "BWF02_FlowRate";
   "Inputs".Level_BWF01 := "BWF01_Level";
   "Inputs".Level_BWF02 := "BWF02_Level";
   "Inputs".TC_01 := "TC01";
   "Inputs".TC_02 := "TC02";
   "Inputs".TC_03 := "TC03";
   "Inputs".TC_06 := "TC06";
   "Inputs".TC_07 := "TC07";
   "Inputs".ZT_01 := "ZT01";
   "Inputs".PSH_01 := "PSH01";
   "Inputs".PSH_02 := "PSH02";
   "Inputs".PSH_03 := "PSH03";
   "Inputs".PC_01 := "PC01";
   "Inputs".FN02_ABSORPTION := "FN02_Current";
   "Inputs".FN04_ABSORPTION := "FN04_Current";
   "Inputs".RD01_ABSORBPTION := "RD01_Current";
   "Inputs".FN01_ABSORPTION := "FN01_Current";
   "Inputs".RO_01 := "R001";
   "Inputs".RO_02 := "R002";
   "Inputs".RO_03 := "R003";
   "Inputs".RO_04 := "R004";
   "Inputs".BR_01_RETRANSMISSION_GAS := "BR01_GAS";
   "Inputs".BR_01_RETRANSMISSION_AIR := "BR01_AIR";
   "Inputs".BR_01_MASSFLOWMETER_GAS := "BR01_FlowMeter_GAS";
   "Inputs".BR_01_MASSFLOWMETER_AIR := "BR01_FlowMeter_AIR";
END_REGION
END_FUNCTION

FUNCTION "HMI PV_1gate" : Void   // FC16, LAD
{ S7_Optimized_Access := 'TRUE' }
VERSION : 0.1
   VAR_INPUT
      LS_Open : Bool;
      LS_Close : Bool;
      Selector : Bool;
      Allarm1 : Bool;
      Allarm2 : Bool;
      Allarm3 : Bool;
      Allarm4 : Bool;
      Allarm5 : Bool;
   END_VAR
   VAR_OUTPUT
      HMI_LS_Open : Bool;
      HMI_LS_Close : Bool;
      Total_Allarms : Bool;
      HMI_Selectoor : Bool;
   END_VAR
BEGIN

REGION Network 1
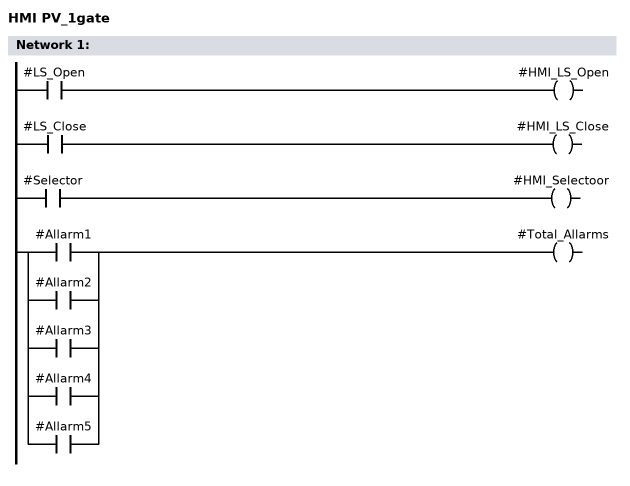
   RUNG wire#powerrail
      Contact( #LS_Open )
      Coil( #HMI_LS_Open )
   END_RUNG
   RUNG wire#powerrail
      Contact( #LS_Close )
      Coil( #HMI_LS_Close )
   END_RUNG
   RUNG wire#powerrail
      Contact( #Selector )
      Coil( #HMI_Selectoor )
   END_RUNG
   RUNG wire#powerrail
      Contact( #Allarm1 )
      wire#w1
      Coil( #Total_Allarms )
   END_RUNG
   RUNG wire#powerrail
      Contact( #Allarm2 )
   END_RUNG wire#w1
   RUNG wire#powerrail
      Contact( #Allarm3 )
   END_RUNG wire#w1
   RUNG wire#powerrail
      Contact( #Allarm4 )
   END_RUNG wire#w1
   RUNG wire#powerrail
      Contact( #Allarm5 )
   END_RUNG wire#w1
   // the same network as SCL:
   #HMI_LS_Open := #LS_Open;
   #HMI_LS_Close := #LS_Close;
   #HMI_Selectoor := #Selector;
   #Total_Allarms := #Allarm1 OR #Allarm2 OR #Allarm3 OR #Allarm4 OR #Allarm5;
END_REGION
END_FUNCTION

FUNCTION "HMI PV_2Gate" : Void   // FC17, LAD
{ S7_Optimized_Access := 'TRUE' }
VERSION : 0.1
   VAR_INPUT
      GateA_Open : Bool;
      GateA_Close : Bool;
      GateB_Open : Bool;
      GateB_Close : Bool;
      Selector_GateA : Bool;
      Selector_GateB : Bool;
      Allarm1 : Bool;
      Allarm2 : Bool;
      Allarm3 : Bool;
      Allarm4 : Bool;
      Allarm5 : Bool;
      Allarm6 : Bool;
      Allarm7 : Bool;
   END_VAR
   VAR_OUTPUT
      HMI_GateA_Open : Bool;
      HMI_GateA_Close : Bool;
      HMI_GateB_Open : Bool;
      HMI_GateB_Close : Bool;
      HMI_Selector_GateA : Bool;
      HMI_Selector_GateB : Bool;
      Total_Allarms : Bool;
   END_VAR
BEGIN

REGION Network 1
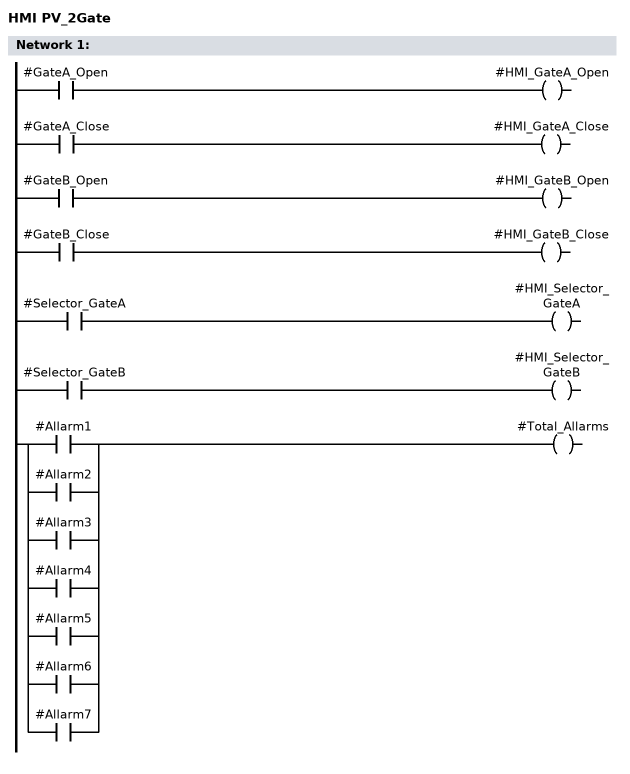
   RUNG wire#powerrail
      Contact( #GateA_Open )
      Coil( #HMI_GateA_Open )
   END_RUNG
   RUNG wire#powerrail
      Contact( #GateA_Close )
      Coil( #HMI_GateA_Close )
   END_RUNG
   RUNG wire#powerrail
      Contact( #GateB_Open )
      Coil( #HMI_GateB_Open )
   END_RUNG
   RUNG wire#powerrail
      Contact( #GateB_Close )
      Coil( #HMI_GateB_Close )
   END_RUNG
   RUNG wire#powerrail
      Contact( #Selector_GateA )
      Coil( #HMI_Selector_GateA )
   END_RUNG
   RUNG wire#powerrail
      Contact( #Selector_GateB )
      Coil( #HMI_Selector_GateB )
   END_RUNG
   RUNG wire#powerrail
      Contact( #Allarm1 )
      wire#w1
      Coil( #Total_Allarms )
   END_RUNG
   RUNG wire#powerrail
      Contact( #Allarm2 )
   END_RUNG wire#w1
   RUNG wire#powerrail
      Contact( #Allarm3 )
   END_RUNG wire#w1
   RUNG wire#powerrail
      Contact( #Allarm4 )
   END_RUNG wire#w1
   RUNG wire#powerrail
      Contact( #Allarm5 )
   END_RUNG wire#w1
   RUNG wire#powerrail
      Contact( #Allarm6 )
   END_RUNG wire#w1
   RUNG wire#powerrail
      Contact( #Allarm7 )
   END_RUNG wire#w1
   // the same network as SCL:
   #HMI_GateA_Open := #GateA_Open;
   #HMI_GateA_Close := #GateA_Close;
   #HMI_GateB_Open := #GateB_Open;
   #HMI_GateB_Close := #GateB_Close;
   #HMI_Selector_GateA := #Selector_GateA;
   #HMI_Selector_GateB := #Selector_GateB;
   #Total_Allarms := #Allarm1 OR #Allarm2 OR #Allarm3 OR #Allarm4 OR #Allarm5 OR #Allarm6 OR #Allarm7;
END_REGION
END_FUNCTION

FUNCTION "HMI Output" : Void   // FC19, LAD
{ S7_Optimized_Access := 'TRUE' }
VERSION : 0.1
BEGIN

REGION Network 1
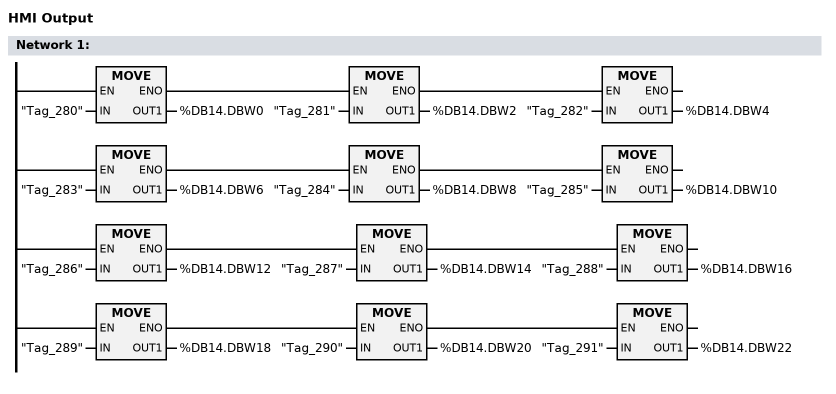
   RUNG wire#powerrail
      Move(in := "Tag_280", out1 => %DB14.DBW0)
      Move(in := "Tag_281", out1 => %DB14.DBW2)
      Move(in := "Tag_282", out1 => %DB14.DBW4)
   END_RUNG
   RUNG wire#powerrail
      Move(in := "Tag_283", out1 => %DB14.DBW6)
      Move(in := "Tag_284", out1 => %DB14.DBW8)
      Move(in := "Tag_285", out1 => %DB14.DBW10)
   END_RUNG
   RUNG wire#powerrail
      Move(in := "Tag_286", out1 => %DB14.DBW12)
      Move(in := "Tag_287", out1 => %DB14.DBW14)
      Move(in := "Tag_288", out1 => %DB14.DBW16)
   END_RUNG
   RUNG wire#powerrail
      Move(in := "Tag_289", out1 => %DB14.DBW18)
      Move(in := "Tag_290", out1 => %DB14.DBW20)
      Move(in := "Tag_291", out1 => %DB14.DBW22)
   END_RUNG
   // the same network as SCL:
   %DB14.DBW0 := "Tag_280";
   %DB14.DBW2 := "Tag_281";
   %DB14.DBW4 := "Tag_282";
   %DB14.DBW6 := "Tag_283";
   %DB14.DBW8 := "Tag_284";
   %DB14.DBW10 := "Tag_285";
   %DB14.DBW12 := "Tag_286";
   %DB14.DBW14 := "Tag_287";
   %DB14.DBW16 := "Tag_288";
   %DB14.DBW18 := "Tag_289";
   %DB14.DBW20 := "Tag_290";
   %DB14.DBW22 := "Tag_291";
END_REGION
END_FUNCTION

FUNCTION "Recipes Handler" : Void   // FC21, SCL
{ S7_Optimized_Access := 'TRUE' }
VERSION : 0.1
   VAR_TEMP
      i : Byte;   // index
      In_Range : Bool;
      Differing : Bool;
   END_VAR
BEGIN
   #In_Range := ("RecipesDB".HMI_Index >= 1 AND "RecipesDB".HMI_Index <= 100);
   #Differing := "RecipesDB".Recipes[0] <> "RecipesDB".Recipes["RecipesDB".HMI_Index];

   //If Hmi editor Idx changes, copy from archvie onto HMI buffer
   IF ("RecipesDB".HMI_Index <> "RecipesDB".OldHmi_Idx) AND #In_Range THEN
       "RecipesDB".Recipes[0] := "RecipesDB".Recipes["RecipesDB".HMI_Index];
       "RecipesDB".Modify_Recipe := 0;
       "RecipesDB".Vis_SaveUndo := 0;
       "RecipesDB".Vis_Modify := 1;
       "RecipesDB".Vis_LoadRecipe := 1;
   //Or if old changed but is not in range, force the first allowed recipe in the editor buffer
   ELSIF NOT #In_Range THEN
       "RecipesDB".HMI_Index := 1;
   END_IF;
   //Changing the hmi idx will force a copy of a new selected recipe on the HMI buffer, no edits are done in the archive.

   //IF HMI Editor idx has NOT changed and is in range, check for modifications between the HMI buffer and the archive copy 
   IF #In_Range AND "RecipesDB".HMI_Index = "RecipesDB".OldHmi_Idx THEN

       //If a modification occured, remove modify button, the operator must save or undo the recipe before proceeding with modifications on other recipes
       //or load any recipes
       IF ("RecipesDB".Recipes[0] <> "RecipesDB".Recipes["RecipesDB".HMI_Index]) AND "RecipesDB".Modify_Recipe THEN
           "RecipesDB".Vis_SaveUndo := 1;
           "RecipesDB".Vis_Modify := 0;
           "RecipesDB".Vis_LoadRecipe := 0;
           //If is possible to save and save btn is pressed, copy editor recipe in archive 
           IF "RecipesDB".Vis_SaveUndo AND "RecipesDB".Save_Recipe THEN
               "RecipesDB".Recipes["RecipesDB".HMI_Index] := "RecipesDB".Recipes[0];
               "RecipesDB".Vis_SaveUndo := 0;
               "RecipesDB".Vis_Modify := 1;
               "RecipesDB".Modify_Recipe:= 0;
               "RecipesDB".Save_Recipe := 0;
               "RecipesDB".Vis_LoadRecipe := 1;
           END_IF;
           //If is possible to undo modification, copy from archive to the editor the recipe
           IF "RecipesDB".Vis_SaveUndo AND "RecipesDB".Undo_Modification THEN
               "RecipesDB".Recipes[0] := "RecipesDB".Recipes["RecipesDB".HMI_Index];
               "RecipesDB".Vis_SaveUndo := 0;
               "RecipesDB".Vis_Modify := 1;
               "RecipesDB".Modify_Recipe := 0;
               "RecipesDB".Undo_Modification := 0;
               "RecipesDB".Vis_LoadRecipe := 1;
           END_IF;
       END_IF;
   END_IF;


   IF ("RecipesDB".Recipes[0] = "RecipesDB".Recipes["RecipesDB".HMI_Index]) AND "RecipesDB".Vis_LoadRecipe AND "RecipesDB".Load_Recipe THEN
       "Data".SET_PERC_BWF01 := "RecipesDB".Recipes[0].BWF01;
       "Data".SET_PERC_BWF02 := "RecipesDB".Recipes[0].BWF02;
       "Data".SET_PERC_FR01 := "RecipesDB".Recipes[0].RD01;
       "Data".SET_PERC_VT01 := "RecipesDB".Recipes[0].FN01;
       "Data".PSH01_SETPOINT := "RecipesDB".Recipes[0].PSH01;
       "Data".PSH02_SETPOINT := "RecipesDB".Recipes[0].PSH02;
       "Data".TC03_SETPOINT := "RecipesDB".Recipes[0].TC03;
       "Data".TC01_SETPOINT := "RecipesDB".Recipes[0].TC01;
       "RecipesDB".Active_Recipe:="RecipesDB".HMI_Index;

       "RecipesDB".Load_Recipe := 0;
   END_IF;



   //Save Last scan Hmi idx
   "RecipesDB".OldHmi_Idx := "RecipesDB".HMI_Index;
END_FUNCTION